INTERFACE ITF_SPM

END_INTERFACE

(* stored: Version 1.1.0.1
   Itf ITF_SPM: Id {f1411ff6-1a67-4fc6-b1c4-cadb1dad2136} *)
